% RSLogix 500 project Final_P3.RSS, saved by version 8.30.00.16 %
PROJECT "UNTITLED"    % processor: Bul.1763 MicroLogix 1100 Series B %

PROGRAM FILES
  LAD 2 "SCAN"  15 rungs
  LAD 3 "LOGIC"  1 rungs

DATA FILES
  O0 OUTPUT  4 elements
  I1 INPUT  6 elements
  S2 STATUS  66 elements
  B3 BINARY  3 elements
  T4 TIMER  1 elements
  C5 COUNTER  1 elements
  R6 CONTROL  1 elements
  N7 INTEGER  10 elements
  F8 FLOAT  1 elements
  ST9 STRING  10 elements
  N10 INTEGER  10 elements
  ST11 STRING  6 elements

LADDER 2 "SCAN"
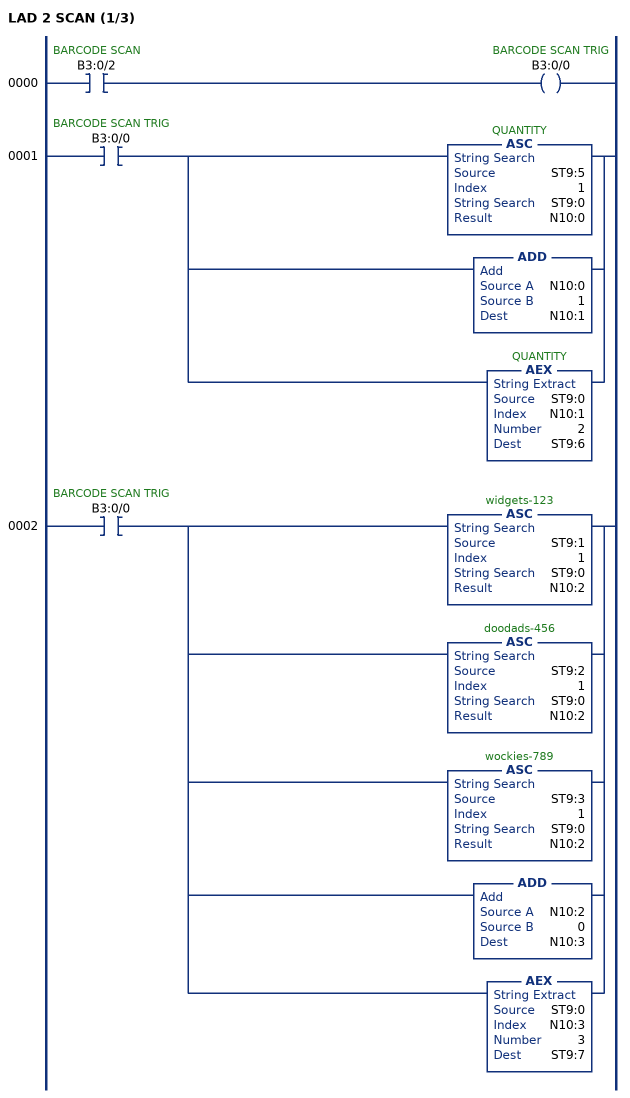
% Rung: 0 %
SOR XIC B3:0/2 OTE B3:0/0 EOR
%   B3:0/2  "BARCODE SCAN" %
%   B3:0/0  "BARCODE SCAN TRIG" %
% Rung: 1 %
SOR XIC B3:0/0 BST ASC ST9:5 1 ST9:0 N10:0 NXB BST ADD N10:0 1 N10:1 NXB AEX ST9:0 N10:1 2 ST9:6 BND BND EOR
%   B3:0/0  "BARCODE SCAN TRIG" %
%   ST9:5  "QUANTITY" %
%   ST9:0  "CODE" %
%   ST9:6  "QUANTITY" %
% Rung: 2 %
SOR XIC B3:0/0 BST BST ASC ST9:1 1 ST9:0 N10:2 NXB BST ASC ST9:2 1 ST9:0 N10:2 NXB ASC ST9:3 1 ST9:0 N10:2 BND BND NXB BST ADD N10:2 0 N10:3 NXB AEX ST9:0 N10:3 3 ST9:7 BND BND EOR
%   B3:0/0  "BARCODE SCAN TRIG" %
%   ST9:1  "widgets-123" %
%   ST9:0  "CODE" %
%   ST9:2  "doodads-456" %
%   ST9:3  "wockies-789" %

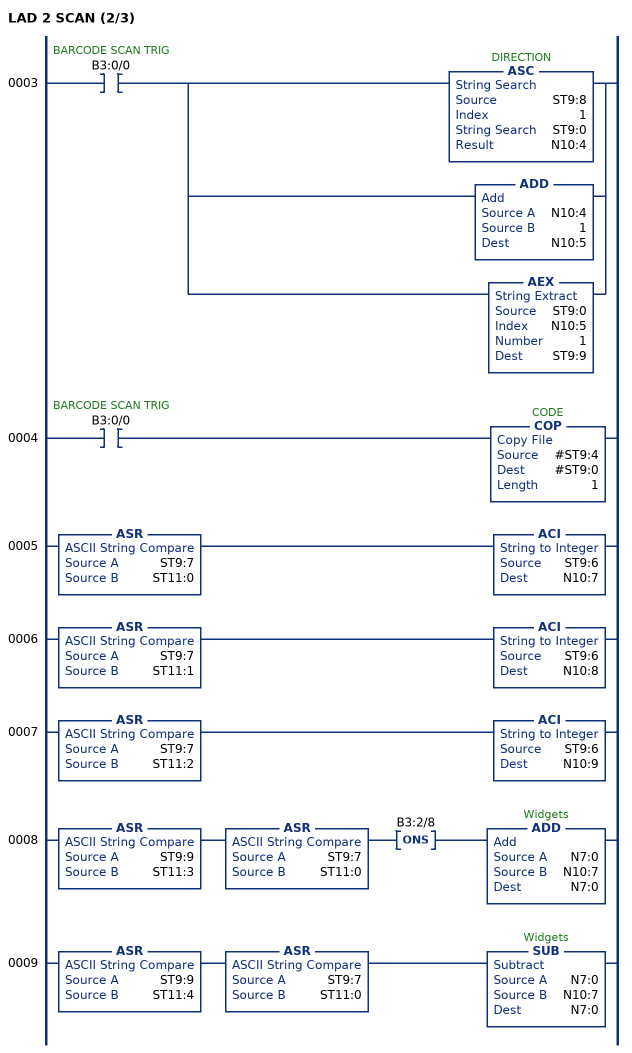
% Rung: 3 %
SOR XIC B3:0/0 BST ASC ST9:8 1 ST9:0 N10:4 NXB BST ADD N10:4 1 N10:5 NXB AEX ST9:0 N10:5 1 ST9:9 BND BND EOR
%   B3:0/0  "BARCODE SCAN TRIG" %
%   ST9:8  "DIRECTION" %
%   ST9:0  "CODE" %
% Rung: 4 %
SOR XIC B3:0/0 COP #ST9:4 #ST9:0 1 EOR
%   B3:0/0  "BARCODE SCAN TRIG" %
%   ST9:4  "CLEAR" %
%   ST9:0  "CODE" %
% Rung: 5 %
SOR ASR ST9:7 ST11:0 ACI ST9:6 N10:7 EOR
%   ST9:6  "QUANTITY" %
% Rung: 6 %
SOR ASR ST9:7 ST11:1 ACI ST9:6 N10:8 EOR
%   ST9:6  "QUANTITY" %
% Rung: 7 %
SOR ASR ST9:7 ST11:2 ACI ST9:6 N10:9 EOR
%   ST9:6  "QUANTITY" %
% Rung: 8 %
SOR ASR ST9:9 ST11:3 ASR ST9:7 ST11:0 ONS B3:2/8 ADD N7:0 N10:7 N7:0 EOR
%   N7:0  "Widgets" %
% Rung: 9 %
SOR ASR ST9:9 ST11:4 ASR ST9:7 ST11:0 SUB N7:0 N10:7 N7:0 EOR
%   N7:0  "Widgets" %

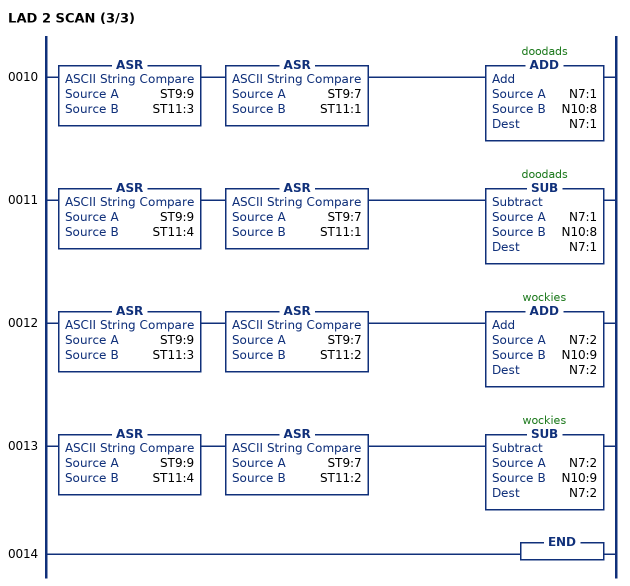
% Rung: 10 %
SOR ASR ST9:9 ST11:3 ASR ST9:7 ST11:1 ADD N7:1 N10:8 N7:1 EOR
%   N7:1  "doodads" %
% Rung: 11 %
SOR ASR ST9:9 ST11:4 ASR ST9:7 ST11:1 SUB N7:1 N10:8 N7:1 EOR
%   N7:1  "doodads" %
% Rung: 12 %
SOR ASR ST9:9 ST11:3 ASR ST9:7 ST11:2 ADD N7:2 N10:9 N7:2 EOR
%   N7:2  "wockies" %
% Rung: 13 %
SOR ASR ST9:9 ST11:4 ASR ST9:7 ST11:2 SUB N7:2 N10:9 N7:2 EOR
%   N7:2  "wockies" %
% Rung: 14 %
SOR END EOR

OTHER DOCUMENTED ADDRESSES
  B3:0/1  "ONE SHOT"
  B3:0/3  "BARCODE RESET"
  B3:0/5  "BARCODE RESET"
  B3:0/6  "ONE SHOT"
  B3:1/0  "ONE SHOT"

DATA TABLE (non-zero values as saved)
DATA ST9
% ST9:0 % "123-10:1"
% ST9:1 % "1"
% ST9:2 % "4"
% ST9:3 % "7"
% ST9:4 % "0"
% ST9:5 % "-"
% ST9:8 % ":"
DATA N10
% N10:0 % 6 7 1 1 0 0 0 0 0 0
DATA ST11
% ST11:0 % "123"
% ST11:1 % "456"
% ST11:2 % "789"
% ST11:3 % "1"
% ST11:4 % "2"
